FUNCTION_BLOCK limit_current
VAR_INPUT
	actual_current : REAL;
	limit_current : REAL;
	th : REAL;
	Enable : BOOL;	
	
	//relief_turn : BOOL := FALSE;	
   
	
END_VAR
VAR_OUTPUT
	Limit_ok :BOOL;
	current : REAL;
END_VAR
VAR
	A : REAL;
	B : REAL;
	
END_VAR


IF Enable = TRUE THEN 
	A := limit_current-th;
	B := limit_current +th;
	
	IF (A <= actual_current) AND (actual_current <= B) THEN 
		current := actual_current;
		IF current >= limit_current THEN
		  Limit_ok := TRUE;			 
		END_IF

	END_IF
ELSE
	 Limit_ok := FALSE;
	
END_IF

END_FUNCTION_BLOCK

(* stored: Version 1.1.0.1, ProductVersion 3.1.4024.4
   POU limit_current: Id {335740a6-22d3-4689-88d6-e65890298b56}, SpecialFunc None *)
